TYPE ST_ZoneData :
(**************************************************************************************
 * 	Application		:	BoxControl Framework
 *	Revision		:	$Revision: 404529 $
 *	Revision date	:	$Date: 2018-04-23 08:21:38 +0200 (Mo., 23 Apr 2018) $
 *	Last changed by	:	$Author: b7bolm $
 *	URL				:	$URL: http://almscdc.swisslog.com/repo/SWPD/Development/BoxControlFramework/20_Release/trunk/01_Software/BCF/BCF/JumpStart/20_Product/10_App/12_E_Functions/10_Lib/10_Conv/01_DUTs/ST_ZoneData.TcDUT $
 *
 *	Purpose			:	Zone data
 *
 * ------------------------------------------------------------------------------------
 *	Copyright Swisslog [IP AG], Switzerland. All rights reserved.
 * 
 * ------------------------------------------------------------------------------------
 *	
 * 	Revision History: 
 *
 * 	VERSION			DATE			INITIALS			DESCRIPTION
 *	0.1				01.01.2001		swl					Example
 *
 **************************************************************************************)
STRUCT
	Init 					: BOOL; // Initialized
	InitRunning				: BOOL; // Initialization running
	AddOn					: ST_AddOnResult; // Valid addon result
	TransportControlData	: ST_TransportControlData; // Transport control data
	ErrorData				: ST_ZoneErrorStruct; // Error structure
	LastTUdata				: ST_LastTUdata; // Data from last TU on position
END_STRUCT
END_TYPE

(* stored: Version 1.1.0.1, ProductVersion 3.1.4024.9
   DUT ST_ZoneData: Id {e41e8b6d-371d-4d21-a653-9ae0b8e02254} *)
